Base_Library.Tracing.Trace.Verbose(MyName, 'Remove a Mover Accepted');
removeMover.Execute(MoverToRemove.IdentInGroup);
FOR i := 0 TO MaxMovers DO
	IF GroupMovers[i] = MoverToRemove THEN
		GroupMovers[i] := 0;
		RegisteredMovers := RegisteredMovers -1;
	END_IF
END_FOR
END_METHOD

METHOD PUBLIC Reset : HRESULT
IF NOT resetCAGroup.Busy THEN
	Base_Library.Tracing.Trace.Verbose(MyName, 'Group Reset Accepted');
	Reset := resetCAGroup.Execute();
END_IF
END_METHOD

END_FUNCTION_BLOCK

// ---- Hardware/NCTController.TcPOU
FUNCTION_BLOCK NCTController EXTENDS CyclicBase
VAR
	_MyInterface: Tc3_XTS_Utility.I_TcIoXtsNctBaseUnitInterface;
END_VAR


//_MyInterface := _MyXpu.NctControllerTcIo().BaseUnitInterfaceTcIo(1);

METHOD Cycle : Base_Library.HRESULT
END_METHOD

PROPERTY MyXtsIoInterface : I_TcIoXtsNctBaseUnitInterface
GET
MyXtsIoInterface := _MyInterface;
END_GET
SET
_MyInterface := MyXtsIoInterface;
END_SET
END_PROPERTY

END_FUNCTION_BLOCK

// ---- Hardware/XTSHardware.TcPOU
FUNCTION_BLOCK XTSHardware EXTENDS CyclicBase IMPLEMENTS I_Initialisable, I_XtsHardware, I_Object
VAR
	XtsParts : ARRAY[0..TcIoXtsEnvironmentParameterList.MaxPartsPerTrack] OF XtsPart('');
	IXtsParts : ARRAY[0..TcIoXtsEnvironmentParameterList.MaxPartsPerTrack] OF XtsPart('');
	_MyNumberParts : INT;
	XtsTracks : ARRAY[0..TcIoXtsEnvironmentParameterList.MaxXtsTracksPerXpu] OF XtsTrack('');
	IXtsTracks : ARRAY[0..TcIoXtsEnvironmentParameterList.MaxXtsTracksPerXpu] OF XtsTrack('');
	_MyNumberTracks : INT;
	TrackOTCIDs: ARRAY [1..Tc3_XTS_Utility.TcIoXtsEnvironmentParameterList.MaxXtsTracksPerXpu] OF Tc3_XTS_Utility.OTCID;
	_MyXpu : Tc3_XTS_Utility.I_TcIoXtsProcessingUnit;
	XtsIoEnvInitialiseState : XtsHardwareInitialisation;
	MyPartCount: UDINT;
	MyTrackCount: UDINT;
	MoverIdDetectionState: MoverIdDetectionStateEnum;
	MoverIdDetectionError: BOOL;
	MoverIdDetected: BOOL;
	_MyXts : INT := 1;
	_MyName : STRING;
	_isInitialised: BOOL;
	_hasXPU : BOOL;
	Status : XtsHardwareStatus;
END_VAR

PROPERTY AllMoverPositionsValid : BOOL
GET
AllMoverPositionsValid := Status.AllMoversValid;
END_GET
END_PROPERTY

PROPERTY AnyPartsInError : BOOL
GET
AnyPartsInError := Status.AreAnyPartsInError;
END_GET
END_PROPERTY

METHOD AreExpectedMoversFound : BOOL
VAR_INPUT
END_VAR
AreExpectedMoversFound := _MyXpu.GetExpectedMoverCount() = _MyXpu.GetDetectedMoverCount();
END_METHOD

METHOD CheckTrackSetForDetection : BOOL
VAR_INPUT
	Track : INT;
END_VAR
CheckTrackSetForDetection := XtsTracks[Track - 1].IsTrackSetForDetection;
END_METHOD

PROPERTY ConfiguredDetectionMoverCount : UDINT
GET
ConfiguredDetectionMoverCount := _MyXpu.GetConfiguredDetectionCount();
END_GET
END_PROPERTY

METHOD PUBLIC  Cycle : HRESULT
VAR
	i : UDINT;
END_VAR
IF NOT _isInitialised THEN
	Cycle := -1;
	RETURN;
END_IF

Status.AllMoversValid := _MyXpu.GetAreAllPositionsValid();
Status.IsInSim :=  _MyXpu.GetOperationMode() = OperationMode.Simulation;
Status.ActiveMoverCount := _MyXpu.GetActiveMoverCount();
Status.AreAllModulesInOp := _MyXpu.GetAreAllModulesInOp();
Status.IsDCLinkVoltageReady := _MyXpu.GetIsDcLinkVoltageReady();
Status.State := _MyXpu.GetDriveState();

Status.AreAnyPartsInError := FALSE;
FOR i := 0 TO TO_INT(MyPartCount - 1) DO
	IF XtsParts[i].HasError THEN
		Status.AreAnyPartsInError := TRUE;
	END_IF
END_FOR

FOR i := 0 TO (MyPartCount - 1) DO
	XtsParts[i].Cycle();
END_FOR
FOR i := 0 TO (MyTrackCount-1) DO
	XtsTracks[i].Cycle();
END_FOR
END_METHOD

PROPERTY DetectedNumberOfParts : INT
GET
DetectedNumberOfParts := TO_INT(_MyNumberParts);
END_GET
END_PROPERTY

PROPERTY DetectedNumberOfTracks : UINT
GET
DetectedNumberOfTracks := TO_UINT( MyTrackCount);
END_GET
END_PROPERTY

PROPERTY ExpectedNumberOfParts : int
GET
ExpectedNumberOfParts := _MyNumberParts;
END_GET
SET
_MyNumberParts := ExpectedNumberOfParts;
END_SET
END_PROPERTY

PROPERTY ExpectedNumberOfTracks : int
GET
ExpectedNumberOfTracks := _MyNumberTracks;
END_GET
SET
_MyNumberTracks := ExpectedNumberOfTracks;
END_SET
END_PROPERTY

METHOD GetPartErrorCode : UDINT
VAR
	i : INT; 
	errorCode : UDINT;
END_VAR
FOR i := 0 TO TO_INT(MyPartCount - 1) DO
	IF XtsParts[i].GetCurrentError() <> 0 THEN
		errorCode := XtsParts[i].GetCurrentError();
		IF errorCode > GetPartErrorCode THEN
			GetPartErrorCode := errorCode;
		END_IF
	END_IF
END_FOR
END_METHOD

METHOD GetTrackInterfaceByNumber : I_XtsTrack
VAR_INPUT
	TrackNumber : UINT;
END_VAR
IF TrackNumber = 0 OR TrackNumber > MyTrackCount THEN
	GetTrackInterfaceByNumber := 0;
	RETURN;
END_IF
GetTrackInterfaceByNumber := XtsTracks[TrackNumber - 1];
END_METHOD

METHOD GetTrackInterfaceByOTCID : I_XtsTrack
VAR_INPUT
	trackOTCID : OTCID;
END_VAR
VAR
	i: INT;
END_VAR
FOR i := 0 TO _MyNumberTracks - 1 DO
	IF trackOTCID = XtsTracks[i].MyOTCID THEN
		GetTrackInterfaceByOTCID := XtsTracks[i];
	END_IF
END_FOR
END_METHOD

METHOD HasValidXPUReference : BOOL
VAR_INPUT
END_VAR
HasValidXPUReference := _hasXPU;
END_METHOD

METHOD Initialise : HRESULT
VAR
	i: INT;
	allInitialised : BOOL;
END_VAR
Initialise := -1;
CASE XtsIoEnvInitialiseState OF
	XtsHardwareInitialisation.WaitingForXpu:
		IF _MyXpu = 0 THEN
			RETURN;
		ELSE
			_MyName := _MyXpu.P_ObjectName;
			XtsIoEnvInitialiseState := XtsHardwareInitialisation.GettingParts;
		END_IF
	XtsHardwareInitialisation.GettingParts:
		MyPartCount := _MyXpu.P_PartCount;
		IF TO_INT(MyPartCount) = _MyNumberParts THEN
			FOR i := 0 TO (TO_INT(MyPartCount) - 1) DO
				XtsParts[i].MyXtsIoEnvInterface := _MyXpu.PartTcIo(TO_UINT(i + 1));
				IXtsParts[i] := XtsParts[i];
				IF THIS^.XtsInSim THEN
					XtsParts[i].SetInSim();
				END_IF
			END_FOR
			XtsIoEnvInitialiseState := XtsHardwareInitialisation.GettingTracks;
		ELSE
			XtsIoEnvInitialiseState := XtsHardwareInitialisation.InitialisationFault;
		END_IF
	XtsHardwareInitialisation.GettingTracks:
		MyTrackCount := _MyXpu.P_TrackCount;
		TrackOTCIDs := _MyXpu.P_TrackOids;
		IF TO_INT(MyTrackCount) = _MyNumberTracks THEN
			FOR i := 0 TO UDINT_TO_INT(MyTrackCount - 1) DO
				XtsTracks[i].MyXtsIoEnvInterface := _MyXpu.TrackTcIo(TO_UINT(i + 1));
				XtsTracks[i].MyOTCID := TrackOTCIDs[i + 1];
				IXtsTracks[i] := XtsTracks[i];
			END_FOR
			XtsIoEnvInitialiseState := XtsHardwareInitialisation.InitialisingXtsParts;
		ELSE
			XtsIoEnvInitialiseState := XtsHardwareInitialisation.InitialisationFault;
		END_IF
	XtsHardwareInitialisation.InitialisingXtsParts:
		allInitialised := TRUE;
		FOR i := 0 TO UDINT_TO_INT(MyPartCount - 1) DO
			IF FAILED(XtsParts[i].Initialise()) THEN
				allInitialised := FALSE;
			END_IF
		END_FOR
		IF allInitialised THEN
			XtsIoEnvInitialiseState := XtsHardwareInitialisation.InitialisingXtsTracks;
		END_IF
	XtsHardwareInitialisation.InitialisingXtsTracks:
		allInitialised := TRUE;
		FOR i := 0 TO UDINT_TO_INT(MyTrackCount - 1) DO
			IF FAILED(XtsTracks[i].Initialise()) THEN
				allInitialised := FALSE;
			END_IF
		END_FOR
		IF allInitialised THEN
			XtsIoEnvInitialiseState := XtsHardwareInitialisation.Initialised;
		END_IF
	XtsHardwareInitialisation.Initialised:
		_isInitialised := TRUE;
		Initialise := 0;
END_CASE
END_METHOD

PROPERTY Initialised : BOOL
GET
Initialised := _isInitialised;
END_GET
END_PROPERTY

METHOD IsHardware24VdcOK : HRESULT
VAR
	i : UDINT;
END_VAR
FOR i := 0 TO (_MyXpu.P_PartCount -1) DO
	IF NOT XtsParts[i].Is24VBusOK() THEN
		IsHardware24VdcOK := -1;
	END_IF
END_FOR
END_METHOD

METHOD IsHardware48VdcOK : HRESULT
VAR
	i : UDINT;
END_VAR
FOR i := 0 TO (_MyXpu.GetPartCount() - 1) DO
	IF NOT XtsParts[i].Is48VBusOK() THEN
		IsHardware48VdcOK := -1;
	END_IF
END_FOR
END_METHOD

METHOD IsIDDetectionStandard : BOOL
VAR_INPUT
END_VAR
IsIDDetectionStandard := _MyXpu.GetMoverIdDetectionMode() = MoverIdDetectionMode.Standard;
END_METHOD

PROPERTY Mover1DetectionState : MoverIdDetectionStateEnum
GET
Mover1DetectionState := _MyXpu.GetMoverIdDetectionState();
END_GET
END_PROPERTY

PROPERTY MoverDetectionState : DetectionStateEnum
GET
MoverDetectionState := _MyXpu.GetDetectionState();
END_GET
END_PROPERTY

PROPERTY MyName : string
GET
MyName := _MyName;
END_GET
END_PROPERTY

PROPERTY MyXpu : I_TcIoXtsProcessingUnit
GET
MyXpu := _MyXpu;
END_GET
SET
_MyXpu := MyXpu;
_hasXPU := TRUE;
END_SET
END_PROPERTY

PROPERTY MyXts : INT
GET
MyXts := _MyXts;
END_GET
SET
_MyXts := MyXts;
END_SET
END_PROPERTY

PROPERTY NumberOfMoversDetected : UDINT
GET
NumberOfMoversDetected := _MyXpu.GetDetectedMoverCount();
END_GET
END_PROPERTY

METHOD RegisterWithParent
VAR_INPUT
	Parent	: I_HostObjects;
END_VAR
Parent.RegisterCyclic(THIS^);
Parent.RegisterInitialisable(THIS^);
END_METHOD

METHOD RemoveATrackFromDetection : HRESULT
VAR_INPUT
	TrackToRemove : UINT;
END_VAR
IF TrackToRemove = 0 THEN
	RemoveATrackFromDetection := -1;
	RETURN;
END_IF
IF TrackToRemove > MyTrackCount THEN
	RemoveATrackFromDetection := -2;
	RETURN;
END_IF
IF MyTrackCount = 1 THEN
	RemoveATrackFromDetection := -3;
	RETURN;
END_IF
XtsTracks[TrackToRemove - 1].RemoveFromDetection();
END_METHOD

METHOD ResetAllParts : BOOL
VAR
	i : INT;
END_VAR
FOR i := 0 TO TO_INT(MyPartCount - 1) DO
	XtsParts[i].ResetPart();
END_FOR
END_METHOD

METHOD ResetAPart : HRESULT
VAR_INPUT
	Part : UINT;
END_VAR
IF Part > MyPartCount THEN
	ResetAPart := -1;
END_IF

IF Part = 0 THEN
	ResetAPart := -2;
END_IF

XtsParts[Part - 1].ResetPart();
END_METHOD

METHOD SetAPartOriginTransform : BOOL
VAR_INPUT
	Part : INT;
	OriginTransform: Tc3_XTS_Utility.ST_OriginTransform;
END_VAR
XtsParts[Part - 1].SetPartOriginTransform(OriginTransform);
END_METHOD

METHOD SetATrackForDetection : HRESULT
VAR_INPUT
	TrackToDetect : UINT;
END_VAR
IF TrackToDetect = 0 THEN
	SetATrackForDetection := -1;
	RETURN;
END_IF
IF TrackToDetect > MyTrackCount THEN
	SetATrackForDetection := -2;
	RETURN;
END_IF

XtsTracks[TrackToDetect - 1].SetForDetection();
END_METHOD

METHOD SetMoverNumberForDetection : HRESULT
VAR_INPUT
	NumberOfMovers : INT;
END_VAR
IF NumberOfMovers < 0 THEN
	SetMoverNumberForDetection := -1;
	RETURN;
END_IF
IF NumberOfMovers > _MyXpu.P_MoverCount THEN
	SetMoverNumberForDetection := -2;
	RETURN;
END_IF
 
_MyXpu.SetConfiguredDetectionCount(nConfiguredMoverDetectionCount := TO_UDINT(NumberOfMovers));
END_METHOD

METHOD TriggerMoverDetection : HRESULT
VAR_INPUT
END_VAR
IF _MyXpu = 0 THEN
	TriggerMoverDetection := -1;
	RETURN;
END_IF
_MyXpu.TriggerDetection();
END_METHOD

METHOD TriggerMoverIDDetection : HRESULT
VAR_INPUT
END_VAR
MoverIdDetectionError 	:= MoverIdDetectionState = MoverIdDetectionStateEnum.Error;
MoverIdDetected 	:= MoverIdDetectionState = MoverIdDetectionStateEnum.Valid;
MoverIdDetectionState	:= _MyXpu.GetMoverIdDetectionState();

IF _MyXpu.GetMoverIdDetectionMode() = MoverIdDetectionMode.Standard THEN
	TriggerMoverIDDetection := -1;
	RETURN;
END_IF
// 
IF MoverIdDetectionState = MoverIdDetectionStateEnum.Running THEN
	TriggerMoverIDDetection := -2;
	RETURN;
END_IF

_MyXpu.TriggerMoverIdDetection();
END_METHOD

METHOD TriggerMoverRedetection : HRESULT
VAR_INPUT
END_VAR
IF _MyXpu = 0 THEN
	TriggerMoverRedetection := -1;
	RETURN;
END_IF

_MyXpu.TriggerRedetection();
END_METHOD

PROPERTY XtsInSim : BOOL
GET
XtsInSim := Status.IsInSim;
END_GET
END_PROPERTY

END_FUNCTION_BLOCK

// ---- Hardware/XtsPart.TcPOU
FUNCTION_BLOCK XtsPart EXTENDS CyclicBase IMPLEMENTS I_Initialisable, I_XtsPart
VAR
	_MyInterface : Tc3_XTS_Utility.I_TcIoXtsXpuPart;
	XtsIoEnvInitialiseState : INT;
	MyModuleCount : UDINT;
	Status : XtsPartStatus;
	MyModules : ARRAY[0..TcIoXtsEnvironmentParameterList.MaxModulesPerPart] OF XtsMotorModule('');
	IMyModules : ARRAY[0..TcIoXtsEnvironmentParameterList.MaxModulesPerPart] OF I_XtsMotorModule;
	ModuleIndex: UDINT := 1;
	CurrentErrorId : UDINT;
	InSim : BOOL;
	PartName: STRING;
	_IsInitialised : BOOL := FALSE;
END_VAR

METHOD PUBLIC  Cycle : HRESULT
VAR
	i : INT;
	tempErrorID : UDINT;
END_VAR
IF _MyInterface = 0 THEN
	Cycle := -1;
	RETURN;
END_IF

Status.PartDriveState := _MyInterface.GetDriveState();
Status.IsDCLinkReady := _MyInterface.GetIsDcLinkVoltageReady();
Status.IsPartActive := _MyInterface.GetIsActive();
Status.PartLength := _MyInterface.GetLength();
Status.AllModuleSsInOP := _MyInterface.GetAreAllModulesInOp();


FOR i := 0 TO (UDINT_TO_UINT(MyModuleCount) - 1) DO
	MyModules[i].Cycle();
END_FOR
END_METHOD

METHOD GetCurrentError : UDINT
VAR_INPUT
END_VAR
GetCurrentError := CurrentErrorId;
END_METHOD

PROPERTY HasError : BOOL
GET
HasError := Status.PartDriveState = DriveState.Fault OR Status.PartDriveState = DriveState.FaultReactionActive OR NOT _MyInterface.GetIsDcLinkVoltageReady();
END_GET
END_PROPERTY

METHOD Initialise : HRESULT
VAR
	i : INT;
END_VAR
Initialise := -1;
CASE XtsIoEnvInitialiseState OF
	0:
		IF _MyInterface <> 0 THEN
			XtsIoEnvInitialiseState := 1;
		ELSE
			XtsIoEnvInitialiseState := 999;
		END_IF
	1:
		MyModuleCount := _MyInterface.P_ModuleCount;
		IF InSim THEN
			XtsIoEnvInitialiseState := 3;
			FOR i := 0 TO UDINT_TO_UINT(MyModuleCount - 1) DO
				MyModules[i].SetInSim();
				IMyModules[i] := MyModules[i];
			END_FOR
			InSim := true;
		ELSE
			FOR i := 0 TO UDINT_TO_UINT(MyModuleCount - 1) DO
				MyModules[i].MyModuleInterface := _MyInterface.ModuleTcIo(i + 1);
				IMyModules[i] := MyModules[i];
			END_FOR
			XtsIoEnvInitialiseState := 2;
		END_IF
		
	2:
		XtsIoEnvInitialiseState := 3;
		FOR i := 0 TO UDINT_TO_UINT(MyModuleCount-1) DO
			IF FAILED(MyModules[i].Initialise()) THEN
				XtsIoEnvInitialiseState := 2;
			END_IF
		END_FOR
	3:
		PartName := _MyInterface.P_ObjectName;
		Initialise := 0;
		_IsInitialised := TRUE;
END_CASE
END_METHOD

PROPERTY Initialised : BOOL
GET
Initialised := _IsInitialised;
END_GET
END_PROPERTY

METHOD Is24VBusOK : BOOL
VAR
	i : INT;
END_VAR
Is24VBusOK := TRUE;
IF NOT InSim THEN
	FOR i := 0 TO (UDINT_TO_UINT(MyModuleCount) - 1) DO
		IF NOT MyModules[i].ControlVdcOK THEN
			Is24VBusOK := FALSE;
		END_IF
	END_FOR
END_IF
END_METHOD

METHOD Is48VBusOK : BOOL
VAR
	i : INT;
END_VAR
Is48VBusOK := TRUE;
IF NOT InSim THEN
	FOR i := 0 TO (UDINT_TO_UINT(MyModuleCount) - 1) DO
		IF NOT MyModules[i].MotorVdcOK THEN
			Is48VBusOK := FALSE;
		END_IF
	END_FOR
END_IF
END_METHOD

PROPERTY MyXtsIoEnvInterface : I_TcIoXtsXpuPart
GET
MyXtsIoEnvInterface := _MyInterface;
END_GET
SET
_MyInterface := MyXtsIoEnvInterface;
END_SET
END_PROPERTY

METHOD ResetPart : BOOL
VAR
	i : INT;
END_VAR
ResetPart := _MyInterface.TriggerReset();
IF NOT InSim THEN
	FOR i := 0 TO (UDINT_TO_UINT(MyModuleCount) - 1) DO
		MyModules[i].AcknowledgeMessages();
	END_FOR
END_IF	
CurrentErrorId := 0;
END_METHOD

METHOD SetInSim : HRESULT
VAR_INPUT
END_VAR
InSim := true;
END_METHOD

METHOD SetPartOriginTransform : BOOL
VAR_INPUT
	OriginTransform: Tc3_XTS_Utility.ST_OriginTransform;
END_VAR
_MyInterface.SetOriginTransform(OriginTransform);
END_METHOD

END_FUNCTION_BLOCK

// ---- Hardware/XtsMotorModule.TcPOU
FUNCTION_BLOCK XtsMotorModule EXTENDS CyclicBase IMPLEMENTS I_Initialisable, I_XtsMotorModule
VAR
	_MyModuleIoInterface : I_TcIoXtsPartModule;
	_IsInitialised : BOOL;
	CurrentLive: LREAL;
	MaxCurrent: LREAL;
	Nominal24Vdc : REAL := 24.0;
	Nominal48Vdc : REAL := 48.0;
	InSim : BOOL;
	Module24Vdc: REAL;
	Module48Vdc: REAL;
	ModuleState: Tc3_XTS_Utility.DriveState;
	ModuleStatus: Tc3_XTS_Utility.CoeStatusInfo;
	ModuleName: STRING;
	MotorOid: OTCID;
	SensorOid: OTCID;
	_BTN: BTN;
	_Infeed : BOOL;
	DiagHistory: ARRAY [1..Tc3_XTS_Utility.TcIoXtsEnvironmentParameterList.MaxDiagMessagesPerModule] OF Tc3_XTS_Utility.DiagHistoryEntry;
	EtherCATState: Tc3_XTS_Utility.EtherCatSlaveStateInfo;
END_VAR

METHOD AcknowledgeMessages : BOOL
VAR_INPUT
END_VAR
IF _MyModuleIoInterface = 0 THEN
	RETURN;
END_IF

AcknowledgeMessages := TRUE;
_MyModuleIoInterface.TriggerAcknowledgeMessages();
END_METHOD

PROPERTY Act24Vdc : LREAL
GET
IF NOT InSim THEN
	Act24Vdc := TO_LREAL(Module24Vdc);
END_IF
END_GET
END_PROPERTY

PROPERTY Act48Vdc : LREAL
GET
IF NOT InSim THEN
	Act48Vdc := Module48Vdc;
END_IF
END_GET
END_PROPERTY

PROPERTY ControlVdcOK : BOOL
GET
ControlVdcOK := TRUE;
IF (Module24Vdc < (Nominal24Vdc * 0.8)) OR (Module24Vdc > (Nominal24Vdc * 1.2)) THEN
	ControlVdcOK := FALSE;
END_IF
END_GET
END_PROPERTY

METHOD PUBLIC  Cycle : HRESULT
VAR_INPUT
END_VAR
VAR
	i : INT;
END_VAR
IF _MyModuleIoInterface = 0 THEN
	Cycle := -1;
	RETURN;
END_IF

IF InSim THEN
	Cycle := -2;
	RETURN;
END_IF

CurrentLive:= _MyModuleIoInterface.GetOverallCurrent();
MaxCurrent:=  _MyModuleIoInterface.GetMaxOverallCurrentLast500ms();
Module24Vdc := _MyModuleIoInterface.GetAuxiliaryVoltage24V();
Module48Vdc := _MyModuleIoInterface.GetDCLinkVoltage();
ModuleState := _MyModuleIoInterface.GetDriveState();
ModuleStatus := _MyModuleIoInterface.GetDriveStatusInfo();
EtherCATState := _MyModuleIoInterface.GetDriveEtherCatSlaveStateInfo();

IF _MyModuleIoInterface.GetHasActiveError() THEN
	DiagHistory := _MyModuleIoInterface.GetLatestMessages();
END_IF
END_METHOD

METHOD Initialise : HRESULT
VAR_INPUT
END_VAR
IF NOT _MyModuleIoInterface.P_IsInitialized THEN
	Initialise := -1;
	RETURN;
END_IF

MotorOid := _MyModuleIoInterface.GetMotorTerminalOid();
SensorOid := _MyModuleIoInterface.GetSensorTerminalOid();
ModuleName := _MyModuleIoInterface.P_ObjectName;
_BTN := _MyModuleIoInterface.GetDriveBTN();
_Infeed := _MyModuleIoInterface.GetIsInfeed();
_IsInitialised := TRUE;
END_METHOD

PROPERTY Initialised : BOOL
GET
Initialised := _IsInitialised;
END_GET
END_PROPERTY

PROPERTY MotorVdcOK : BOOL
GET
MotorVdcOK := TRUE;
IF (Module48Vdc < (Nominal48Vdc * 0.8)) OR (Module48Vdc > (Nominal48Vdc * 1.2)) THEN
	MotorVdcOK := FALSE;
END_IF
END_GET
END_PROPERTY

PROPERTY MyModuleInterface : I_TcIoXtsPartModule
GET
MyModuleInterface := _MyModuleIoInterface;
END_GET
SET
_MyModuleIoInterface := MyModuleInterface;
END_SET
END_PROPERTY

METHOD SetInSim : HRESULT
VAR_INPUT
END_VAR
InSim := true;
END_METHOD

END_FUNCTION_BLOCK
